# EPICS autosave request: elveFlowApp/Db/elveFlow_settings.req
$(P)$(R)Pres1
$(P)$(R)P1TweakVal
$(P)$(R)OB1sensorType
